FUNCTION_BLOCK HmiEnableDisableAllVisitor IMPLEMENTS I_ComponentVisitor, I_ModuleVisitor
VAR
	{attribute 'hide'}
	HmiFunction : I_HmiFunction;
	{attribute 'hide'}
	Enable : BOOL;
END_VAR

METHOD DisableHmi
VAR_INPUT
	Module : I_Module;
END_VAR
Enable := FALSE;
Module.Accept(THIS^);
END_METHOD

METHOD EnableHmi
VAR_INPUT
	Module : I_Module;
END_VAR
Enable := TRUE;
Module.Accept(THIS^);
END_METHOD

METHOD VisitComponent
VAR_INPUT
	Component : I_Component;
END_VAR
IF __QUERYINTERFACE(Component, HmiFunction) THEN
	IF Enable THEN
		HmiFunction.Enable();
	ELSE
		HmiFunction.Disable();
	END_IF
END_IF
END_METHOD

METHOD VisitModule
VAR_INPUT
	Module : I_Module;
END_VAR
Module.Components.Accept(THIS^);
Module.Modules.Accept(THIS^);
END_METHOD

END_FUNCTION_BLOCK

(* stored: Version 1.1.0.1, ProductVersion 3.1.4026.18
   POU HmiEnableDisableAllVisitor: Id {cfb5fe83-b725-45b3-9067-bf9c9aa81124}, SpecialFunc None
   Method DisableHmi: Id {5f27f88f-92fc-4b4b-96b5-8d1cd4d91220}
   Method EnableHmi: Id {3d907a07-a549-418e-9c97-c3b4a2dd5177}
   Method VisitComponent: Id {4ab272de-4b42-4f91-8d46-a400c7576a86}
   Method VisitModule: Id {2883ee86-0aac-4f37-bfe5-dcdf254a93bf} *)
